// TwinCAT 3 PLC project TcPiper
// Title: TcPiper
// Company: Loupe
// Author: Loupe
// ProjectVersion: 0.0.4
// ProgramVersion: 3.1.4024.0
// libraries:
//   Tc2_Standard, * (Beckhoff Automation GmbH)
//   Tc2_System, * (Beckhoff Automation GmbH)
//   Tc3_Module, * (Beckhoff Automation GmbH)
//   TcCommando, * (Loupe)
//   TcPluginFramework, * (Loupe)
//   TcSequencer, * (Loupe)
//   TcUnit, * (www.tcunit.org)
// project tree:
//   DUTs/ MACHINE_STATE.TcTLEO, RESPONSE_STATE.TcTLEO
//   GVLs/ PIPER_CONST.TcGVL
//   PiperModule/ IPiperModule.TcIO, PiperImplements.TcDUT, PiperModule.TcPOU, PiperModuleInternal.TcDUT
//   Piper/ GroupStatus.TcPOU, Piper.TcPOU, PiperCommand.TcDUT, PiperStatus.TcDUT, PiperSubmoduleCollection.TcDUT
//   / PlcTask.TcTTO
//   Test/ PiperModule_Test.TcPOU, Piper_Test.TcPOU, TESTPRG.TcPOU
//   Test/Instances/ Piper_EM.TcPOU, TaskFB.TcPOU (not stored)
// real-time tasks:
//   TASK PlcTask: cycle T#10ms, priority 20, ADS port 350

CONFIGURATION TcPiper
    RESOURCE PLC ON TwinCAT3
        TASK PlcTask(INTERVAL := T#10ms, PRIORITY := 20);
        PROGRAM TESTPRG WITH PlcTask : TESTPRG;
    END_RESOURCE
END_CONFIGURATION

// ---- DUTs/MACHINE_STATE.TcTLEO
{attribute 'qualified_only'}
{attribute 'strict'}
{attribute 'to_string'}
TYPE MACHINE_STATE :
(
	BOOTING := 0,
	ABORTING,
	ABORTED,
	CLEARING,
	COMPLETING, 
	COMPLETE, 
	EXECUTING,
	HOLDING,
	HELD,
	IDLE,
	RESETTING,
	STARTING,
	STOPPING,
	STOPPED,
	SUSPENDING,
	SUSPENDED,
	UNHOLDING,
	UNSUSPENDING,
	END	
);
END_TYPE

// ---- DUTs/RESPONSE_STATE.TcTLEO
{attribute 'qualified_only'}
{attribute 'strict'}
TYPE RESPONSE_STATE :
(
	UNDEFINED,
	BUSY,
	DONE,
	DONE_PENDING,
	SUBSTATE,
	ERROR,
	NO_IMPL
);
END_TYPE

// ---- PiperModule/PiperImplements.TcDUT
TYPE
    PiperImplements :
    STRUCT
        aborting : BOOL;
        booting : BOOL;
        clearing : BOOL;
        completing : BOOL;
        executing : BOOL;
        holding : BOOL;
        resetting : BOOL;
        starting : BOOL;
        stopping : BOOL;
        suspending : BOOL;
        unholding : BOOL;
        unsuspending : BOOL;
    END_STRUCT
END_TYPE

// ---- PiperModule/PiperModuleInternal.TcDUT
TYPE
    PiperModuleInternal :
    STRUCT
        machine : REFERENCE TO Piper;
        context : IPluginRunner;
        registered : BOOL;
        response : RESPONSE_STATE;
        requestSubstate : ULINT;
        previousSubstate : ULINT;
        previousSubstateAsync : ULINT;
        skipsSync : PiperImplements;
        skipsAsync : PiperImplements;
        requestNumber : DINT;
    END_STRUCT
END_TYPE

// ---- Piper/PiperCommand.TcDUT
TYPE
    PiperCommand :
    STRUCT
        Abort : BOOL;
        Start : BOOL;
        Stop : BOOL;
        Clear : BOOL;
        Reset : BOOL;
        Suspend : BOOL;
        Unsuspend : BOOL;
        Hold : BOOL;
        Unhold : BOOL;
    END_STRUCT
END_TYPE;

// ---- Piper/PiperStatus.TcDUT
TYPE
    PiperStatus :
    STRUCT
        state : MACHINE_STATE;
        subState : DINT;
    END_STRUCT
END_TYPE

// ---- Piper/PiperSubmoduleCollection.TcDUT
TYPE
    PiperSubmoduleCollection :
    STRUCT
        countSubmodules : INT;
        submodules : ARRAY[0..MAI_NUM_PIPER_MODULES] OF IPiperModule;
        busyModules : ARRAY[0..MAI_NUM_PIPER_MODULES] OF IPiperModule;
        errorModules : ARRAY[0..MAI_NUM_PIPER_MODULES] OF IPiperModule;
        doneModules : ARRAY[0..MAI_NUM_PIPER_MODULES] OF IPiperModule;
    END_STRUCT
END_TYPE

// ---- GVLs/PIPER_CONST.TcGVL
VAR_GLOBAL CONSTANT
    MAX_NUM_PIPER_MODULES : USINT := 100;
    MAI_NUM_PIPER_MODULES : USINT := MAX_NUM_PIPER_MODULES - 1;
END_VAR

// ---- PiperModule/IPiperModule.TcIO
INTERFACE IPiperModule EXTENDS IPlugin
// Copyright (c) 2024 Loupe (https://loupe.team), provided under the MIT License.

METHOD Aborting : MACHINE_STATE
END_METHOD

METHOD AbortingAsync : MACHINE_STATE
END_METHOD

METHOD Booting : MACHINE_STATE
END_METHOD

METHOD BootingAsync : MACHINE_STATE
END_METHOD

METHOD CallState : BOOL
VAR_INPUT

END_VAR
END_METHOD

METHOD CallStateAsync : BOOL
VAR_INPUT
END_VAR
END_METHOD

METHOD Clearing : MACHINE_STATE
END_METHOD

METHOD ClearingAsync : MACHINE_STATE
END_METHOD

METHOD Completing : MACHINE_STATE
END_METHOD

METHOD CompletingAsync : MACHINE_STATE
END_METHOD

PROPERTY CurrentState : MACHINE_STATE
GET
END_GET
END_PROPERTY

METHOD DidCall : BOOL
VAR_INPUT
END_VAR
END_METHOD

METHOD DidCallAsync : BOOL
VAR_INPUT
END_VAR
END_METHOD

METHOD Executing : MACHINE_STATE
END_METHOD

METHOD ExecutingAsync : MACHINE_STATE
END_METHOD

METHOD Holding : MACHINE_STATE
END_METHOD

METHOD HoldingAsync : MACHINE_STATE
END_METHOD

METHOD RegisterToMachine : DINT
VAR_INPUT
    machineIn : REFERENCE TO Piper;
END_VAR
END_METHOD

{warning 'add property implementation'}
PROPERTY RequestedSubstate : ULINT
GET
END_GET
END_PROPERTY

METHOD Resetting : BOOL
END_METHOD

METHOD ResettingAsync : BOOL
END_METHOD

PROPERTY Response : RESPONSE_STATE
GET
END_GET
END_PROPERTY

METHOD Run : BOOL
END_METHOD

METHOD SetContext : BOOL
VAR_INPUT
    context : IPluginRunner;
END_VAR
END_METHOD

METHOD SetState : BOOL
VAR_INPUT
END_VAR
END_METHOD

METHOD Starting : MACHINE_STATE
END_METHOD

METHOD StartingAsync : MACHINE_STATE
END_METHOD

METHOD Stopping : MACHINE_STATE
END_METHOD

METHOD StoppingAsync : MACHINE_STATE
END_METHOD

METHOD Suspending : MACHINE_STATE
END_METHOD

METHOD SuspendingAsync : MACHINE_STATE
END_METHOD

METHOD Undefined : MACHINE_STATE
END_METHOD

METHOD UndefinedAsync : MACHINE_STATE
END_METHOD

METHOD Unholding : MACHINE_STATE
END_METHOD

METHOD UnholdingAsync : MACHINE_STATE
END_METHOD

METHOD Unsuspending : MACHINE_STATE
END_METHOD

METHOD UnsuspendingAsync : MACHINE_STATE
END_METHOD

METHOD WillCall : BOOL
VAR_INPUT
END_VAR
END_METHOD

METHOD WillCallAsync : BOOL
VAR_INPUT
END_VAR
END_METHOD

END_INTERFACE

// ---- Test/TESTPRG.TcPOU
PROGRAM TESTPRG
VAR
    piperTest : Piper_Test;
    piperModuleTest : PiperModule_Test;
END_VAR

// Copyright (c) 2024 Loupe (https://loupe.team), provided under the MIT License.

TcUnit.RUN();

END_PROGRAM

// ---- Test/Piper_Test.TcPOU
FUNCTION_BLOCK Piper_Test EXTENDS FB_TestSuite
VAR_INPUT
END_VAR
VAR_OUTPUT
END_VAR
VAR
END_VAR

// Copyright (c) 2024 Loupe (https://loupe.team), provided under the MIT License.

CommandSetsState();
StateTransitions();

METHOD AbortAndClear
VAR_INPUT
    piper : REFERENCE TO Piper;
END_VAR
// Copyright (c) 2024 Loupe (https://loupe.team), provided under the MIT License.

piper.command.Abort := TRUE;
piper();
AssertEquals_DINT(piper.packMLState, MACHINE_STATE.ABORTING, Message := 'State should be ABORTING');
piper.NextState();
AssertEquals_DINT(piper.packMLState, MACHINE_STATE.ABORTED, Message := 'State after STARTING should be ABORTED');

piper.command.Clear := TRUE;
piper();
AssertEquals_DINT(piper.packMLState, MACHINE_STATE.CLEARING, Message := 'State should be CLEARING');
piper.NextState();
AssertEquals_DINT(piper.packMLState, MACHINE_STATE.STOPPED, Message := 'State after CLEARING should be STOPPED');
END_METHOD

METHOD CommandSetsState
VAR
    piper : Piper;
END_VAR
// Copyright (c) 2024 Loupe (https://loupe.team), provided under the MIT License.

// Check that state actually gets set
// Run this sanity check before the full state transition checks
TEST('SetState');
piper.command.Reset := TRUE;
piper();
AssertFalse(piper.command.Reset, Message := 'Command should be cyclicly reset');
AssertEquals_DINT(piper.packMLState,
    MACHINE_STATE.RESETTING,
    Message := 'Setting a valid state command and cyclic calling FUB once should change state');

TEST_FINISHED();
END_METHOD

METHOD Holding : BOOL
VAR_INPUT
    piper : REFERENCE TO Piper;
END_VAR
// Copyright (c) 2024 Loupe (https://loupe.team), provided under the MIT License.

piper.command.Hold := TRUE;
piper();
AssertEquals_DINT(Expected := piper.packMLState, Actual := MACHINE_STATE.HOLDING, Message := 'State should be HOLDING');
END_METHOD

METHOD Resetting
VAR_INPUT
    piper : REFERENCE TO Piper;
END_VAR
// Copyright (c) 2024 Loupe (https://loupe.team), provided under the MIT License.

piper.command.Reset := TRUE;
piper();
AssertEquals_DINT(Expected := piper.packMLState, Actual := MACHINE_STATE.RESETTING, Message := 'State should be RESETTING');
END_METHOD

METHOD StartAndExecute : BOOL
VAR_INPUT
    piper : REFERENCE TO Piper;
END_VAR
// Copyright (c) 2024 Loupe (https://loupe.team), provided under the MIT License.

piper.command.Start := TRUE;
piper();
AssertEquals_DINT(piper.packMLState, MACHINE_STATE.STARTING, Message := 'State should be STARTING');
piper.NextState();
piper();
END_METHOD

METHOD Starting
VAR_INPUT
    piper : REFERENCE TO Piper;
END_VAR
// Copyright (c) 2024 Loupe (https://loupe.team), provided under the MIT License.

piper.command.Start := TRUE;
piper();
AssertEquals_DINT(piper.packMLState, MACHINE_STATE.STARTING, Message := 'State should be STARTING');
END_METHOD

METHOD StateTransitions
VAR
    piper : Piper();
    task : TaskFB();
    piperModule : Piper_EM(piper, task);
END_VAR
// Copyright (c) 2024 Loupe (https://loupe.team), provided under the MIT License.

// This test confirms the order of state progressions per PackML (with additional BOOTING state)
// With no submodules, it's expected Piper will proceed immediately to the next state

(*STweep.Disable*)

TEST('BootAndReset');
	// Note: there is currently no abort while booting
	AssertEquals_DINT(piper.packMLState, MACHINE_STATE.BOOTING, Message := 'Initil state should be BOOTING');
	piper.NextState();
	AssertEquals_DINT(piper.packMLState, MACHINE_STATE.STOPPED, Message := 'STOPPED state should be after BOOTING');
	
	Resetting(piper);
	piper.NextState();
	AssertEquals_DINT(piper.packMLState, MACHINE_STATE.IDLE, Message := 'Next state after RESETTING should be IDLE');

TEST_FINISHED();

TEST('StartAndAbortWhileStarting');
	Starting(piper);
	
	AbortAndClear(piper);
	
	Resetting(piper);
	piper.NextState();
	AssertEquals_DINT(piper.packMLState, MACHINE_STATE.IDLE, Message := 'Next state after RESETTING should be IDLE');
TEST_FINISHED();

TEST('ResetAndAbortWhileResetting');
	AbortAndClear(piper); // Get into CLEARED
	Resetting(piper);
	// in resetting
	AbortAndClear(piper);
	// stopped
	Resetting(piper);
	piper.NextState();
	AssertEquals_DINT(piper.packMLState, MACHINE_STATE.IDLE, Message := 'Next state after RESETTING should be IDLE');
TEST_FINISHED();

TEST('ExecuteAndAbortWhileExecuting');
	Starting(piper);
	piper.NextState(); // in Executing
	AbortAndClear(piper);
	// stopped
	Resetting(piper);
	piper.NextState();
	AssertEquals_DINT(piper.packMLState, MACHINE_STATE.IDLE, Message := 'Next state after RESETTING should be IDLE');
TEST_FINISHED();

TEST('ExecuteAndStop');
	Starting(piper);
	piper.NextState(); // in Executing
	
	Stopping(piper);
	piper.NextState();
	// stopped
	Resetting(piper);
	piper.NextState();
	AssertEquals_DINT(piper.packMLState, MACHINE_STATE.IDLE, Message := 'Next state after RESETTING should be IDLE');
TEST_FINISHED();

//TEST('HoldAndUnhold');
//	piper.RegisterSubmodule(piperModule);
//	Starting(piper);
//	piper.NextState(); // in Executing

//	Holding(piper);
//	Unholding(piper);

//	Stopping(piper);
//	piper.NextState();
//	// stopped
//	Resetting(piper);
//	piper.NextState();
//	AssertEquals_DINT(piper.PackMLState, MACHINE_STATE.IDLE, Message := 'Next state after RESETTING should be IDLE');
//TEST_FINISHED();

//TEST('SuspendAndUnSuspend');
//	Starting(piper);
//	piper.NextState(); // in Executing

//	Suspending(piper);
//	Unsuspending(piper);

//	Stopping(piper);
//	piper.NextState();
//	// stopped
//	Resetting(piper);
//	piper.NextState();
//	AssertEquals_DINT(piper.PackMLState, MACHINE_STATE.IDLE, Message := 'Next state after RESETTING should be IDLE');
//TEST_FINISHED();
END_METHOD

METHOD Stopping : BOOL
VAR_INPUT
    piper : REFERENCE TO Piper;
END_VAR
// Copyright (c) 2024 Loupe (https://loupe.team), provided under the MIT License.

piper.command.Stop := TRUE;
piper();
AssertEquals_DINT(piper.packMLState, MACHINE_STATE.STOPPING, Message := 'State should be STOPPING');
END_METHOD

METHOD Suspending : BOOL
VAR_INPUT
    piper : REFERENCE TO Piper;
END_VAR
// Copyright (c) 2024 Loupe (https://loupe.team), provided under the MIT License.

piper.command.Suspend := TRUE;
piper();
AssertEquals_DINT(Expected := piper.packMLState, Actual := MACHINE_STATE.SUSPENDING, Message := 'State should be SUSPENDING');
END_METHOD

METHOD Unholding : BOOL
VAR_INPUT
    piper : REFERENCE TO Piper;
END_VAR
// Copyright (c) 2024 Loupe (https://loupe.team), provided under the MIT License.

piper.command.Unhold := TRUE;
piper();
AssertEquals_DINT(Expected := piper.packMLState, Actual := MACHINE_STATE.UNHOLDING, Message := 'State should be UNHOLDING');
END_METHOD

METHOD Unsuspending : BOOL
VAR_INPUT
    piper : REFERENCE TO Piper;
END_VAR
// Copyright (c) 2024 Loupe (https://loupe.team), provided under the MIT License.

piper.command.Unsuspend := TRUE;
piper();
AssertEquals_DINT(Expected := piper.packMLState, Actual := MACHINE_STATE.UNSUSPENDING, Message := 'State should be UNSUSPENDING');
END_METHOD

END_FUNCTION_BLOCK

// ---- Piper/Piper.TcPOU
FUNCTION_BLOCK Piper
VAR_INPUT
    command : PiperCommand;
END_VAR
VAR_OUTPUT
    packMLState : MACHINE_STATE;
END_VAR
VAR
    _substate : ULINT;
    submodules : PiperSubmoduleCollection;
END_VAR

// Copyright (c) 2024 Loupe (https://loupe.team), provided under the MIT License.

UpdateSystemState();
HandleBoolCommands();
CallCurrentState();

METHOD CallCurrentState : MACHINE_STATE
VAR_INPUT
END_VAR
VAR
    i : INT;
    currentModule : IPiperModule;
END_VAR
// Copyright (c) 2024 Loupe (https://loupe.team), provided under the MIT License.

FOR i := 0 TO submodules.countSubmodules - 1 DO

    currentModule := submodules.submodules[i];
    currentModule.CallStateAsync();

END_FOR
END_METHOD

METHOD HandleBoolCommands : BOOL
VAR_INPUT
END_VAR
// Copyright (c) 2024 Loupe (https://loupe.team), provided under the MIT License.

//Standard state transitions
CASE packMLState OF
    MACHINE_STATE.ABORTED:
        IF command.Clear THEN
            SetState(MACHINE_STATE.CLEARING);
        END_IF

    MACHINE_STATE.STOPPED:
        IF command.Reset THEN
            SetState(MACHINE_STATE.RESETTING);
        END_IF

    MACHINE_STATE.COMPLETE:
        IF command.Reset THEN
            SetState(MACHINE_STATE.RESETTING);
        END_IF

    MACHINE_STATE.IDLE:
        IF command.Start THEN
            SetState(MACHINE_STATE.STARTING);
        END_IF

    MACHINE_STATE.HELD:
        IF command.Unhold THEN
            SetState(MACHINE_STATE.UNHOLDING);
        END_IF

    MACHINE_STATE.SUSPENDED:
        IF command.Unsuspend THEN
            SetState(MACHINE_STATE.UNSUSPENDING);
        END_IF

END_CASE

//Stop state transitions
//Can happen in all states except stop/ing and abort/ing 
CASE packMLState OF
    MACHINE_STATE.STOPPED,
        MACHINE_STATE.STOPPING,
        MACHINE_STATE.ABORTED,
        MACHINE_STATE.ABORTING:
        ;
ELSE
    IF command.Stop THEN
        SetState(MACHINE_STATE.STOPPING);
    END_IF
END_CASE

//Abort state transitions
//Can happen in all states except abort/ing 
CASE packMLState OF
    MACHINE_STATE.ABORTED,
        MACHINE_STATE.ABORTING:
        ;
ELSE
    IF command.Abort THEN
        SetState(MACHINE_STATE.ABORTING);
    END_IF
END_CASE

command.Abort := FALSE;
command.Clear := FALSE;
command.Hold := FALSE;
command.Reset := FALSE;
command.Start := FALSE;
command.Stop := FALSE;
command.Suspend := FALSE;
command.Unhold := FALSE;
command.Unsuspend := FALSE;
END_METHOD

METHOD NextState
VAR_INPUT
END_VAR
// Copyright (c) 2024 Loupe (https://loupe.team), provided under the MIT License.

CASE packMLState OF
    MACHINE_STATE.ABORTING:
        SetState(MACHINE_STATE.ABORTED);

    MACHINE_STATE.BOOTING:
        SetState(MACHINE_STATE.STOPPED);

    MACHINE_STATE.CLEARING:
        SetState(MACHINE_STATE.STOPPED);

    MACHINE_STATE.COMPLETING:
        SetState(MACHINE_STATE.COMPLETE);

    MACHINE_STATE.EXECUTING:
        SetState(MACHINE_STATE.COMPLETE);

    MACHINE_STATE.RESETTING:
        SetState(MACHINE_STATE.IDLE);

    MACHINE_STATE.HOLDING:
        SetState(MACHINE_STATE.HELD);

    MACHINE_STATE.STARTING:
        SetState(MACHINE_STATE.EXECUTING);

    MACHINE_STATE.STOPPING:
        SetState(MACHINE_STATE.STOPPED);

    MACHINE_STATE.SUSPENDING:
        SetState(MACHINE_STATE.SUSPENDED);

    MACHINE_STATE.UNHOLDING:
        SetState(MACHINE_STATE.EXECUTING);

    MACHINE_STATE.UNSUSPENDING:
        SetState(MACHINE_STATE.EXECUTING);

END_CASE
END_METHOD

METHOD PackMLStateIsTransition : BOOL
VAR_INPUT
END_VAR
// Copyright (c) 2024 Loupe (https://loupe.team), provided under the MIT License.

packMLStateIsTransition :=
    packMLState = MACHINE_STATE.ABORTING OR
    packMLState = MACHINE_STATE.BOOTING OR
    packMLState = MACHINE_STATE.CLEARING OR
    packMLState = MACHINE_STATE.COMPLETING OR
    packMLState = MACHINE_STATE.EXECUTING OR
    packMLState = MACHINE_STATE.HOLDING OR
    packMLState = MACHINE_STATE.RESETTING OR
    packMLState = MACHINE_STATE.STARTING OR
    packMLState = MACHINE_STATE.STOPPING OR
    packMLState = MACHINE_STATE.SUSPENDING OR
    packMLState = MACHINE_STATE.UNHOLDING OR
    packMLState = MACHINE_STATE.UNSUSPENDING;
END_METHOD

METHOD RegisterSubmodule : UDINT
VAR_INPUT
    subsystem : IPiperModule;
END_VAR
// Copyright (c) 2024 Loupe (https://loupe.team), provided under the MIT License.

IF submodules.countSubmodules < MAI_NUM_PIPER_MODULES THEN
    submodules.submodules[submodules.countSubmodules] := subsystem;
    submodules.countSubmodules := submodules.countSubmodules + 1;
END_IF
END_METHOD

METHOD PRIVATE SetState : BOOL
VAR_INPUT
    state : MACHINE_STATE;
END_VAR
VAR
    i : INT;
    currentModule : IPiperModule;
END_VAR
// Copyright (c) 2024 Loupe (https://loupe.team), provided under the MIT License.

packMLState := state;

Substate := 0;

FOR i := 0 TO submodules.countSubmodules - 1 DO

    currentModule := submodules.submodules[i];

    currentModule.SetState();

END_FOR
END_METHOD

PROPERTY Substate : ULINT
GET
// Copyright (c) 2024 Loupe (https://loupe.team), provided under the MIT License.

Substate := _substate;
END_GET
SET
// Copyright (c) 2024 Loupe (https://loupe.team), provided under the MIT License.

_substate := Substate;
END_SET
END_PROPERTY

METHOD UpdateSystemState : BOOL
VAR_INPUT
END_VAR

VAR
    i : INT;
    currentModule : IPiperModule;
    busy : INT;
    error : INT;
    done : INT;
    substateRequest : ULINT;
END_VAR
VAR CONSTANT
    maxULINT : ULINT := -1;
END_VAR
// Copyright (c) 2024 Loupe (https://loupe.team), provided under the MIT License.

busy := 0;
done := 0;
error := 0;

FOR i := 0 TO MAI_NUM_PIPER_MODULES DO
    submodules.busyModules[i] := 0;
    submodules.doneModules[i] := 0;
    submodules.errorModules[i] := 0;
    //	IF NOT Submodules.submodules[i].hasContext THEN
    //TODO: 	REFUSE TO RUN AND THROW ERROR
    //			MSG: add FB_Init with THIS^.setContext(Synchronous Context);		
    //	END_IF
END_FOR

substateRequest := maxULINT;

IF packMLStateIsTransition() THEN

    FOR i := 0 TO submodules.countSubmodules - 1 DO
        currentModule := submodules.submodules[i];

        CASE currentModule.Response OF
            RESPONSE_STATE.UNDEFINED,
                RESPONSE_STATE.BUSY:
                submodules.busyModules[busy] := currentModule;

                // If the module is requesting a substate, it isn't busy, it's waiting
                IF currentModule.RequestedSubstate <> 0 THEN

                    // If it is requesting a lower substate than what is currently being requested
                    // it wins and should be called next
                    IF currentModule.RequestedSubstate < substateRequest AND currentModule.RequestedSubstate > Substate THEN

                        substateRequest := currentModule.RequestedSubstate;

                    ELSIF currentModule.RequestedSubstate = Substate THEN

                        busy := busy + 1;

                    END_IF
                ELSE
                    busy := busy + 1;
                END_IF

            RESPONSE_STATE.DONE_PENDING,
                RESPONSE_STATE.DONE:
                submodules.doneModules[done] := currentModule;
                done := done + 1;

            RESPONSE_STATE.ERROR:
                submodules.errorModules[error] := currentModule;
                error := error + 1;

        END_CASE
    END_FOR

END_IF

//If there are errors, we go to aborting, unless we are already aborting..
IF error > 0 THEN

    IF packMLState <> MACHINE_STATE.ABORTING THEN
        SetState(MACHINE_STATE.ABORTING);
    END_IF

ELSIF busy = 0 THEN

    IF substateRequest < maxULINT AND substateRequest > Substate THEN
        Substate := substateRequest;
    ELSE
        nextState();
    END_IF
    //ELSIF  THEN

END_IF
END_METHOD

END_FUNCTION_BLOCK

// ---- PiperModule/PiperModule.TcPOU
FUNCTION_BLOCK ABSTRACT PiperModule IMPLEMENTS IPiperModule, ISequence, IStepManager
VAR
    _piperModule : PiperModuleInternal;
    _sequence : SequenceType;
    _sequencer : Sequencer(THIS^);
	
    command : PLCopenCall;
END_VAR

// Copyright (c) 2024 Loupe (https://loupe.team), provided under the MIT License.

METHOD _RequestStep : BOOL
VAR_INPUT
    nextStep : ENUM;
END_VAR
// Copyright (c) 2024 Loupe (https://loupe.team), provided under the MIT License.

_piperModule.requestSubstate := nextStep;
_piperModule.response := RESPONSE_STATE.BUSY;
_piperModule.requestNumber := _piperModule.requestNumber + 1;
END_METHOD

METHOD _Reset : BOOL
// Copyright (c) 2024 Loupe (https://loupe.team), provided under the MIT License.
END_METHOD

METHOD _SequenceComplete : BOOL
// Copyright (c) 2024 Loupe (https://loupe.team), provided under the MIT License.

_piperModule.requestSubstate := 0;
_piperModule.response := RESPONSE_STATE.DONE;
END_METHOD

METHOD _SequenceError : BOOL
// Copyright (c) 2024 Loupe (https://loupe.team), provided under the MIT License.

_piperModule.requestSubstate := 0;
_piperModule.response := RESPONSE_STATE.ERROR;
END_METHOD

METHOD Aborted : BOOL
// Copyright (c) 2024 Loupe (https://loupe.team), provided under the MIT License.

_sequence.activeTasks.Aborted();
END_METHOD

METHOD Aborting : MACHINE_STATE
// Copyright (c) 2024 Loupe (https://loupe.team), provided under the MIT License.

_piperModule.skipsSync.aborting := TRUE;
END_METHOD

METHOD AbortingAsync : MACHINE_STATE
// Copyright (c) 2024 Loupe (https://loupe.team), provided under the MIT License.

_piperModule.skipsAsync.aborting := TRUE;
END_METHOD

METHOD Booting : MACHINE_STATE
// Copyright (c) 2024 Loupe (https://loupe.team), provided under the MIT License.

_piperModule.skipsSync.booting := TRUE;
END_METHOD

METHOD BootingAsync : MACHINE_STATE
// Copyright (c) 2024 Loupe (https://loupe.team), provided under the MIT License.

_piperModule.skipsAsync.booting := TRUE;
END_METHOD

METHOD CallState : BOOL
VAR_INPUT

END_VAR
// Copyright (c) 2024 Loupe (https://loupe.team), provided under the MIT License.

THIS^.WillCall();

IF THIS^._piperModule.previousSubstate <> THIS^.CurrentSubstate THEN
    THIS^.WillChangeSubstate();
END_IF

THIS^._piperModule.previousSubstate := THIS^.CurrentSubstate;

IF Response <> RESPONSE_STATE.DONE AND RequestedSubstate <= CurrentSubstate THEN
    CASE CurrentState OF
        MACHINE_STATE.ABORTING:
            IF NOT _piperModule.skipsSync.aborting THEN
                THIS^.Aborting();
            END_IF

        MACHINE_STATE.BOOTING:
            IF NOT _piperModule.skipsSync.booting THEN
                THIS^.Booting();
            END_IF

        MACHINE_STATE.CLEARING:
            IF NOT _piperModule.skipsSync.clearing THEN
                THIS^.Clearing();
            END_IF

        MACHINE_STATE.COMPLETING:
            IF NOT _piperModule.skipsSync.completing THEN
                THIS^.COMPLETING();
            END_IF

        MACHINE_STATE.EXECUTING:
            IF NOT _piperModule.skipsSync.executing THEN
                THIS^.Executing();
            END_IF

        MACHINE_STATE.HOLDING:
            IF NOT _piperModule.skipsSync.holding THEN
                THIS^.Holding();
            END_IF

        MACHINE_STATE.RESETTING:
            IF NOT _piperModule.skipsSync.resetting THEN
                THIS^.Resetting();
            END_IF

        MACHINE_STATE.STARTING:
            IF NOT _piperModule.skipsSync.starting THEN
                THIS^.Starting();
            END_IF

        MACHINE_STATE.STOPPING:
            IF NOT _piperModule.skipsSync.stopping THEN
                THIS^.Stopping();
            END_IF

        MACHINE_STATE.SUSPENDING:
            IF NOT _piperModule.skipsSync.suspending THEN
                THIS^.Suspending();
            END_IF

        MACHINE_STATE.UNHOLDING:
            IF NOT _piperModule.skipsSync.unholding THEN
                THIS^.Unholding();
            END_IF

        MACHINE_STATE.UNSUSPENDING:
            IF NOT _piperModule.skipsSync.unsuspending THEN
                THIS^.Unsuspending();
            END_IF

    END_CASE
END_IF

THIS^.DidCall();
END_METHOD

METHOD CallStateAsync : BOOL
VAR_INPUT

END_VAR
// Copyright (c) 2024 Loupe (https://loupe.team), provided under the MIT License.

THIS^.WillCallAsync();

IF THIS^._piperModule.previousSubstateAsync <> THIS^.CurrentSubstate THEN
    THIS^.WillChangeSubstateAsync();
END_IF

THIS^._piperModule.previousSubstateAsync := THIS^.CurrentSubstate;

IF Response <> RESPONSE_STATE.DONE AND RequestedSubstate <= CurrentSubstate THEN
    CASE CurrentState OF
        MACHINE_STATE.ABORTING:
            IF NOT _piperModule.skipsAsync.aborting THEN
                THIS^.AbortingAsync();
            ELSIF _piperModule.skipsSync.aborting THEN
                _piperModule.response := RESPONSE_STATE.DONE;
            END_IF

        MACHINE_STATE.BOOTING:
            IF NOT _piperModule.skipsAsync.booting THEN
                THIS^.BootingAsync();
            ELSIF _piperModule.skipsSync.booting THEN
                _piperModule.response := RESPONSE_STATE.DONE;
            END_IF

        MACHINE_STATE.CLEARING:
            IF NOT _piperModule.skipsAsync.clearing THEN
                THIS^.ClearingAsync();
            ELSIF _piperModule.skipsSync.clearing THEN
                _piperModule.response := RESPONSE_STATE.DONE;
            END_IF

        MACHINE_STATE.COMPLETING:
            IF NOT _piperModule.skipsAsync.completing THEN
                THIS^.CompletingAsync();
            ELSIF _piperModule.skipsSync.completing THEN
                _piperModule.response := RESPONSE_STATE.DONE;
            END_IF

        MACHINE_STATE.EXECUTING:
            IF NOT _piperModule.skipsAsync.executing THEN
                THIS^.ExecutingAsync();
            ELSIF _piperModule.skipsSync.executing THEN
                _piperModule.response := RESPONSE_STATE.DONE;
            END_IF

        MACHINE_STATE.HOLDING:
            IF NOT _piperModule.skipsAsync.holding THEN
                THIS^.HoldingAsync();
            ELSIF _piperModule.skipsSync.holding THEN
                _piperModule.response := RESPONSE_STATE.DONE;
            END_IF

        MACHINE_STATE.RESETTING:
            IF NOT _piperModule.skipsAsync.resetting THEN
                THIS^.ResettingAsync();
            ELSIF _piperModule.skipsSync.resetting THEN
                _piperModule.response := RESPONSE_STATE.DONE;
            END_IF

        MACHINE_STATE.STARTING:
            IF NOT _piperModule.skipsAsync.starting THEN
                THIS^.StartingAsync();
            ELSIF _piperModule.skipsSync.starting THEN
                _piperModule.response := RESPONSE_STATE.DONE;
            END_IF

        MACHINE_STATE.STOPPING:
            IF NOT _piperModule.skipsAsync.stopping THEN
                THIS^.StoppingAsync();
            ELSIF _piperModule.skipsSync.stopping THEN
                _piperModule.response := RESPONSE_STATE.DONE;
            END_IF

        MACHINE_STATE.SUSPENDING:
            IF NOT _piperModule.skipsAsync.suspending THEN
                THIS^.SuspendingAsync();
            ELSIF _piperModule.skipsSync.suspending THEN
                _piperModule.response := RESPONSE_STATE.DONE;
            END_IF

        MACHINE_STATE.UNHOLDING:
            IF NOT _piperModule.skipsAsync.unholding THEN
                THIS^.UnholdingAsync();
            ELSIF _piperModule.skipsSync.unholding THEN
                _piperModule.response := RESPONSE_STATE.DONE;
            END_IF

        MACHINE_STATE.UNSUSPENDING:
            IF NOT _piperModule.skipsAsync.unsuspending THEN
                THIS^.UnsuspendingAsync();
            ELSIF _piperModule.skipsSync.unsuspending THEN
                _piperModule.response := RESPONSE_STATE.DONE;
            END_IF

    END_CASE
END_IF

THIS^.DidCallAsync();
END_METHOD

METHOD PRIVATE CheckStatus : BOOL
VAR
    _commandIndex : INT;
    _anyAbort : BOOL;
    _anyBusy : BOOL;
    _anyError : BOOL;
END_VAR
// Copyright (c) 2024 Loupe (https://loupe.team), provided under the MIT License.

IF NOT _sequence.statusChecked THEN
    //We cache the is abort so that we have a consistent 
    //	status for the whole state
    _sequence.isError := _sequence.activeTasks.isError;
    _sequence.isAbort := _sequence.activeTasks.isAbort;
    _sequence.isDone := _sequence.activeTasks.isDone;
END_IF
END_METHOD

METHOD Clearing : MACHINE_STATE
// Copyright (c) 2024 Loupe (https://loupe.team), provided under the MIT License.

_piperModule.skipsSync.clearing := TRUE;
END_METHOD

METHOD ClearingAsync : MACHINE_STATE
// Copyright (c) 2024 Loupe (https://loupe.team), provided under the MIT License.

_piperModule.skipsAsync.clearing := TRUE;
END_METHOD

METHOD Completing : MACHINE_STATE
// Copyright (c) 2024 Loupe (https://loupe.team), provided under the MIT License.

_piperModule.skipsSync.completing := TRUE;
END_METHOD

METHOD CompletingAsync : MACHINE_STATE
// Copyright (c) 2024 Loupe (https://loupe.team), provided under the MIT License.

_piperModule.skipsAsync.completing := TRUE;
END_METHOD

PROPERTY CurrentState : MACHINE_STATE
GET
// Copyright (c) 2024 Loupe (https://loupe.team), provided under the MIT License.

CurrentState := _piperModule.machine.packMLState;
END_GET
END_PROPERTY

PROPERTY CurrentStep : ENUM
GET
// Copyright (c) 2024 Loupe (https://loupe.team), provided under the MIT License.

CurrentStep := ULINT_TO_UDINT(_piperModule.machine.Substate);
END_GET
END_PROPERTY

PROPERTY CurrentSubstate : ULINT
GET
// Copyright (c) 2024 Loupe (https://loupe.team), provided under the MIT License.

CurrentSubstate := _piperModule.machine.Substate;
END_GET
END_PROPERTY

METHOD DidCall : BOOL
VAR_INPUT
END_VAR
// Copyright (c) 2024 Loupe (https://loupe.team), provided under the MIT License.
END_METHOD

METHOD DidCallAsync : BOOL
VAR_INPUT
END_VAR
// Copyright (c) 2024 Loupe (https://loupe.team), provided under the MIT License.
END_METHOD

METHOD DoStep : ENUM
VAR
END_VAR
// Copyright (c) 2024 Loupe (https://loupe.team), provided under the MIT License.

DoStep := _sequencer.DoStep();
END_METHOD

METHOD Errored : BOOL
VAR_INPUT
    ID : INT;
END_VAR
// Copyright (c) 2024 Loupe (https://loupe.team), provided under the MIT License.

_sequence.activeTasks.Errored(ID);
END_METHOD

METHOD Executing : MACHINE_STATE
// Copyright (c) 2024 Loupe (https://loupe.team), provided under the MIT License.

_piperModule.skipsSync.executing := TRUE;
END_METHOD

METHOD ExecutingAsync : MACHINE_STATE
// Copyright (c) 2024 Loupe (https://loupe.team), provided under the MIT License.

_piperModule.skipsAsync.executing := TRUE;
END_METHOD

METHOD FB_init : BOOL
VAR_INPUT
    bInitRetains : BOOL; // if TRUE, the retain variables are initialized (warm start / cold start)
    bInCopyCode : BOOL; // if TRUE, the instance afterwards gets moved into the copy code (online change)
    machineIn : REFERENCE TO Piper;
    //	context : IPluginRunner;
END_VAR
// Copyright (c) 2024 Loupe (https://loupe.team), provided under the MIT License.
RegisterToMachine(machineIn);
//THIS^.setContext( context );
END_METHOD

METHOD Finished : BOOL
// Copyright (c) 2024 Loupe (https://loupe.team), provided under the MIT License.

_sequence.activeTasks.Finished();
END_METHOD

METHOD Holding : MACHINE_STATE
// Copyright (c) 2024 Loupe (https://loupe.team), provided under the MIT License.

_piperModule.skipsSync.holding := TRUE;
END_METHOD

METHOD HoldingAsync : MACHINE_STATE
// Copyright (c) 2024 Loupe (https://loupe.team), provided under the MIT License.

_piperModule.skipsAsync.holding := TRUE;
END_METHOD

PROPERTY IsAbort : BOOL
GET
// Copyright (c) 2024 Loupe (https://loupe.team), provided under the MIT License.

CheckStatus();
IsAbort := _sequence.isAbort;
END_GET
END_PROPERTY

PROPERTY IsDone : BOOL
GET
// Copyright (c) 2024 Loupe (https://loupe.team), provided under the MIT License.

CheckStatus();
IsDone := _sequence.isDone;
END_GET
END_PROPERTY

PROPERTY IsError : BOOL
GET
// Copyright (c) 2024 Loupe (https://loupe.team), provided under the MIT License.

CheckStatus();
IsError := _sequence.isError;
END_GET
END_PROPERTY

METHOD OnAbort : BOOL
VAR_INPUT
    nextStep : ENUM;
END_VAR
// Copyright (c) 2024 Loupe (https://loupe.team), provided under the MIT License.

OnAbort := _sequencer.OnAbort(nextStep);
END_METHOD

METHOD OnEntry : BOOL
VAR_INPUT
END_VAR
// Copyright (c) 2024 Loupe (https://loupe.team), provided under the MIT License.

OnEntry := _sequencer.OnEntry();
END_METHOD

METHOD OnError : BOOL
VAR_INPUT
    nextStep : ENUM;
END_VAR
// Copyright (c) 2024 Loupe (https://loupe.team), provided under the MIT License.

OnError := _sequencer.OnError(nextStep);
END_METHOD

METHOD OnExit : BOOL
VAR_INPUT
END_VAR
// Copyright (c) 2024 Loupe (https://loupe.team), provided under the MIT License.

OnExit := _sequencer.OnExit();
END_METHOD

METHOD OnFailure : BOOL
VAR_INPUT
    nextStep : ENUM;
END_VAR
// Copyright (c) 2024 Loupe (https://loupe.team), provided under the MIT License.

OnFailure := _sequencer.OnFailure(nextStep);
END_METHOD

METHOD OnSuccess : BOOL
VAR_INPUT
    nextStep : ENUM;
END_VAR
// Copyright (c) 2024 Loupe (https://loupe.team), provided under the MIT License.

OnSuccess := _sequencer.OnSuccess(nextStep);
END_METHOD

METHOD RegisterToMachine : DINT
VAR_INPUT
    machineIn : REFERENCE TO Piper;
END_VAR
VAR
END_VAR
// Copyright (c) 2024 Loupe (https://loupe.team), provided under the MIT License.
IF NOT _piperModule.registered THEN
    _piperModule.registered := TRUE;
    _piperModule.machine REF= machineIn;
    _piperModule.machine.RegisterSubmodule(THIS^);
END_IF
END_METHOD

{warning 'add property implementation'}
PROPERTY RequestedSubstate : ULINT
GET
// Copyright (c) 2024 Loupe (https://loupe.team), provided under the MIT License.

RequestedSubstate := _piperModule.requestSubstate;
END_GET
END_PROPERTY

PROPERTY RequestNumber : DINT
GET
// Copyright (c) 2024 Loupe (https://loupe.team), provided under the MIT License.

RequestNumber := _piperModule.requestNumber;
END_GET
END_PROPERTY

METHOD RequestStep : BOOL
VAR_INPUT
    nextStep : ENUM;
END_VAR
// Copyright (c) 2024 Loupe (https://loupe.team), provided under the MIT License.

RequestStep := _sequencer.requestStep(nextStep);
END_METHOD

METHOD RequestStepClear : BOOL
VAR_INPUT
    nextStep : ENUM;
END_VAR
// Copyright (c) 2024 Loupe (https://loupe.team), provided under the MIT License.

RequestStepClear := _sequencer.requestStepClear(nextStep);
END_METHOD

METHOD Resetting : BOOL
// Copyright (c) 2024 Loupe (https://loupe.team), provided under the MIT License.

_piperModule.skipsSync.resetting := TRUE;
END_METHOD

METHOD ResettingAsync : BOOL
// Copyright (c) 2024 Loupe (https://loupe.team), provided under the MIT License.

_piperModule.skipsAsync.resetting := TRUE;
END_METHOD

PROPERTY Response : RESPONSE_STATE
GET
// Copyright (c) 2024 Loupe (https://loupe.team), provided under the MIT License.

Response := _piperModule.response;
END_GET
END_PROPERTY

METHOD Run : BOOL
// Copyright (c) 2024 Loupe (https://loupe.team), provided under the MIT License.

THIS^.CallState();
END_METHOD

METHOD SequenceAbort : BOOL
VAR_INPUT
    ErrorCode : DINT;
    ErrorMessage : STRING;
END_VAR
// Copyright (c) 2024 Loupe (https://loupe.team), provided under the MIT License.

SequenceAbort := _sequencer.sequenceAbort(ErrorCode, ErrorMessage);
END_METHOD

METHOD SequenceComplete : BOOL
VAR_INPUT
END_VAR
// Copyright (c) 2024 Loupe (https://loupe.team), provided under the MIT License.

SequenceComplete := _sequencer.sequenceComplete();
END_METHOD

METHOD SequenceError : BOOL
VAR_INPUT
    ErrorCode : DINT;
    ErrorMessage : STRING;
END_VAR
// Copyright (c) 2024 Loupe (https://loupe.team), provided under the MIT License.

SequenceError := _sequencer.sequenceError(ErrorCode, ErrorMessage);
END_METHOD

METHOD SetContext : BOOL
VAR_INPUT
    context : IPluginRunner;
END_VAR
// Copyright (c) 2024 Loupe (https://loupe.team), provided under the MIT License.
_piperModule.context := context;
context.RegisterPlugin(THIS^);
END_METHOD

METHOD SetState : BOOL
VAR_INPUT
END_VAR
// Copyright (c) 2024 Loupe (https://loupe.team), provided under the MIT License.

_piperModule.requestSubstate := 0;
_piperModule.response := RESPONSE_STATE.UNDEFINED;
_sequencer.startSequence();
END_METHOD

METHOD Start : BOOL
VAR_INPUT
    Command : IPLCopenCommand;
END_VAR
// Copyright (c) 2024 Loupe (https://loupe.team), provided under the MIT License.

IF _sequence.activeTasks.Start(Command) = 0 THEN
    //TODO: All out of commands.. Throw an error
    SequenceError(10000, 'Too Many Commands in 1 step');
    Start := FALSE;
ELSE
    Start := TRUE;
END_IF
END_METHOD

METHOD Starting : MACHINE_STATE
// Copyright (c) 2024 Loupe (https://loupe.team), provided under the MIT License.

_piperModule.skipsSync.starting := TRUE;
END_METHOD

METHOD StartingAsync : MACHINE_STATE
// Copyright (c) 2024 Loupe (https://loupe.team), provided under the MIT License.

_piperModule.skipsAsync.starting := TRUE;
END_METHOD

METHOD StartSequence : BOOL
// Copyright (c) 2024 Loupe (https://loupe.team), provided under the MIT License.

RequestStep(0);
END_METHOD

METHOD StateCompletePending : BOOL
VAR_INPUT
END_VAR
// Copyright (c) 2024 Loupe (https://loupe.team), provided under the MIT License.

_piperModule.response := RESPONSE_STATE.DONE_PENDING;
END_METHOD

METHOD StateErrored : BOOL
VAR_INPUT
END_VAR
// Copyright (c) 2024 Loupe (https://loupe.team), provided under the MIT License.

_piperModule.response := RESPONSE_STATE.ERROR;
END_METHOD

METHOD Stopping : MACHINE_STATE
// Copyright (c) 2024 Loupe (https://loupe.team), provided under the MIT License.

_piperModule.skipsSync.stopping := TRUE;
END_METHOD

METHOD StoppingAsync : MACHINE_STATE
// Copyright (c) 2024 Loupe (https://loupe.team), provided under the MIT License.

_piperModule.skipsAsync.stopping := TRUE;
END_METHOD

METHOD Suspending : MACHINE_STATE
// Copyright (c) 2024 Loupe (https://loupe.team), provided under the MIT License.

_piperModule.skipsSync.suspending := TRUE;
END_METHOD

METHOD SuspendingAsync : MACHINE_STATE
// Copyright (c) 2024 Loupe (https://loupe.team), provided under the MIT License.

_piperModule.skipsAsync.suspending := TRUE;
END_METHOD

METHOD Undefined : MACHINE_STATE
// Copyright (c) 2024 Loupe (https://loupe.team), provided under the MIT License.

_piperModule.response := RESPONSE_STATE.NO_IMPL;
END_METHOD

METHOD UndefinedAsync : MACHINE_STATE
// Copyright (c) 2024 Loupe (https://loupe.team), provided under the MIT License.
END_METHOD

METHOD Unholding : MACHINE_STATE
// Copyright (c) 2024 Loupe (https://loupe.team), provided under the MIT License.

_piperModule.skipsSync.unholding := TRUE;
END_METHOD

METHOD UnholdingAsync : MACHINE_STATE
// Copyright (c) 2024 Loupe (https://loupe.team), provided under the MIT License.

_piperModule.skipsAsync.unholding := TRUE;
END_METHOD

METHOD Unsuspending : MACHINE_STATE
// Copyright (c) 2024 Loupe (https://loupe.team), provided under the MIT License.

_piperModule.skipsSync.unsuspending := TRUE;
END_METHOD

METHOD UnsuspendingAsync : MACHINE_STATE
// Copyright (c) 2024 Loupe (https://loupe.team), provided under the MIT License.

_piperModule.skipsAsync.unsuspending := TRUE;
END_METHOD

METHOD WillCall : BOOL
VAR_INPUT
END_VAR
// Copyright (c) 2024 Loupe (https://loupe.team), provided under the MIT License.
END_METHOD

METHOD WillCallAsync : BOOL
VAR_INPUT
END_VAR
// Copyright (c) 2024 Loupe (https://loupe.team), provided under the MIT License.
END_METHOD

METHOD WillChangeSubstate : BOOL
VAR_INPUT
END_VAR
// Copyright (c) 2024 Loupe (https://loupe.team), provided under the MIT License.
END_METHOD

METHOD WillChangeSubstateAsync : BOOL
VAR_INPUT
END_VAR
// Copyright (c) 2024 Loupe (https://loupe.team), provided under the MIT License.
END_METHOD

END_FUNCTION_BLOCK

// ---- Test/Instances/Piper_EM.TcPOU
FUNCTION_BLOCK Piper_EM EXTENDS PiperModule
VAR_INPUT
END_VAR
VAR_OUTPUT
END_VAR
VAR
    task : REFERENCE TO TaskFB;
    keepExecuting : BOOL := TRUE;
END_VAR

// Copyright (c) 2024 Loupe (https://loupe.team), provided under the MIT License.

METHOD Executing : MACHINE_STATE
// Copyright (c) 2024 Loupe (https://loupe.team), provided under the MIT License.

WHILE keepExecuting DO
    ;
    //
END_WHILE
END_METHOD

METHOD FB_init : BOOL
VAR_INPUT
    bInitRetains : BOOL; // if TRUE, the retain variables are initialized (warm start / cold start)
    bInCopyCode : BOOL; // if TRUE, the instance afterwards gets moved into the copy code (online change)
    machineIn : REFERENCE TO Piper;
    taskFB : REFERENCE TO TaskFB;
    //	context : IPluginRunner;
END_VAR
// Copyright (c) 2024 Loupe (https://loupe.team), provided under the MIT License.

THIS^.SetContext(taskFB);
task REF= taskFB;
END_METHOD

END_FUNCTION_BLOCK

// ---- Test/PiperModule_Test.TcPOU
FUNCTION_BLOCK PiperModule_Test EXTENDS FB_TestSuite
VAR_INPUT
END_VAR
VAR_OUTPUT
END_VAR
VAR
END_VAR

// Copyright (c) 2024 Loupe (https://loupe.team), provided under the MIT License.

END_FUNCTION_BLOCK

// ---- Piper/GroupStatus.TcPOU
FUNCTION_BLOCK GroupStatus
VAR_INPUT
END_VAR
VAR_OUTPUT
END_VAR
VAR
    _Busy : BOOL;
    _Error : BOOL;
END_VAR

// Copyright (c) 2024 Loupe (https://loupe.team), provided under the MIT License.

METHOD Busy
VAR_INPUT
    Message : STRING[80];
END_VAR
// Copyright (c) 2024 Loupe (https://loupe.team), provided under the MIT License.

_Busy := TRUE;
END_METHOD

METHOD Error
VAR_INPUT
    Message : STRING[80];
END_VAR
// Copyright (c) 2024 Loupe (https://loupe.team), provided under the MIT License.

_Error := TRUE;
END_METHOD

PROPERTY IsBusy : BOOL
GET
// Copyright (c) 2024 Loupe (https://loupe.team), provided under the MIT License.

IsBusy := NOT _Error AND _Busy;
END_GET
END_PROPERTY

PROPERTY IsDone : BOOL
GET
// Copyright (c) 2024 Loupe (https://loupe.team), provided under the MIT License.

IsDone := NOT _Error AND NOT _Busy;
END_GET
END_PROPERTY

PROPERTY IsError : BOOL
GET
// Copyright (c) 2024 Loupe (https://loupe.team), provided under the MIT License.

IsError := _Error;
END_GET
END_PROPERTY

METHOD Ok : BOOL
VAR_INPUT
END_VAR
// Copyright (c) 2024 Loupe (https://loupe.team), provided under the MIT License.
END_METHOD

METHOD Reset
VAR_INPUT
END_VAR
// Copyright (c) 2024 Loupe (https://loupe.team), provided under the MIT License.

_Busy := FALSE;
_Error := FALSE;
END_METHOD

PROPERTY Status : PLCopenStatusBase
GET
// Copyright (c) 2024 Loupe (https://loupe.team), provided under the MIT License.

IF _Error THEN

    Status := PLCopenStatusBase.ERROR;

ELSIF _Busy THEN

    Status := PLCopenStatusBase.BUSY;

ELSE

    Status := PLCopenStatusBase.ERR_OK;

END_IF
END_GET
END_PROPERTY

END_FUNCTION_BLOCK
